// TwinCAT 3 PLC project Untitled1
// ProgramVersion: 3.1.4026.1+972e9c44872ad038b353624a861fd7e3244e9f75
// libraries:
//   Tc2_Standard, * (Beckhoff Automation GmbH)
//   Tc2_System, * (Beckhoff Automation GmbH)
//   Tc2_Utilities, * (Beckhoff Automation GmbH)
// project tree:
//   GVLs/ GVL.TcGVL
//   / PlcTask.TcTTO
//   POUs/ MAIN.TcPOU, ReadingFile.TcPOU, WritingFile.TcPOU
// real-time tasks:
//   TASK PlcTask: cycle T#10ms, priority 20, ADS port 350

CONFIGURATION Untitled1
    RESOURCE PLC ON TwinCAT3
        TASK PlcTask(INTERVAL := T#10ms, PRIORITY := 20);
        PROGRAM MAIN WITH PlcTask : MAIN;
    END_RESOURCE
END_CONFIGURATION

// ---- GVLs/GVL.TcGVL
{attribute 'qualified_only'}
VAR_GLOBAL
	sPath : STRING := 'C:\SampleFile\Test.txt';
	
END_VAR

// ---- POUs/MAIN.TcPOU
PROGRAM MAIN
VAR
	
END_VAR

ReadingFile();
WritingFile();

END_PROGRAM

// ---- POUs/ReadingFile.TcPOU
PROGRAM ReadingFile
VAR
	fbFileOpen : FB_FileOpen;
	fbFileRead : FB_FileRead;
	fbFileClose : FB_FileClose;
	hFile : UINT;
	sRead : T_MAXSTRING;
	bStartRead : BOOL;
	bReset : BOOL;
	
	eState : (init, FileOpen, FileRead, FileClose, TextFileToString , StringToINT , Error);
	i : INT;
	
	NewLineCount : INT;
	sTemp : ARRAY[1..MAX_LENGTH] OF STRING;
	nINT : ARRAY[1..MAX_LENGTH] OF INT;
	nTemp : INT;
END_VAR

VAR CONSTANT
	MAX_LENGTH : INT := 20;
END_VAR

CASE eState OF
	init :
		IF bStartRead THEN
			bStartRead := FALSE;
			eState := FileOpen;
		END_IF
		
	FileOpen :
		fbFileOpen(
			sPathName:= GVL.sPath, 
			nMode:= FOPEN_MODEREAD OR FOPEN_MODETEXT, 
			bExecute:= TRUE, 
			hFile=> hFile);
		IF NOT fbFileOpen.bBusy THEN
			IF fbFileOpen.bError THEN
				eState := Error;
			ELSE
				eState := FileRead;
				MEMSET(ADR(sRead), 0, SIZEOF(sRead) );
			END_IF
			fbFileOpen(bExecute := FALSE);
		END_IF
		
	FileRead : //fbFileRead로 값을 읽어 sRead에 값을 입력
		fbFileRead(
			hFile:= hFile, 
			pReadBuff:=ADR(sRead) , 
			cbReadLen:= SIZEOF(sRead), 
			bExecute:= TRUE);
		IF NOT fbFileRead.bBusy THEN
			IF fbFileRead.bError THEN
				eState := Error;
			ELSE
				eState := FileClose;
			END_IF
			fbFileRead(bExecute := FALSE);
		END_IF
	
	FileClose :
		fbFileClose(
			hFile:= hFile, 
			bExecute:= TRUE);
		IF NOT fbFileClose.bBusy THEN
			IF fbFileClose.bError THEN
				eState := Error;
			ELSE
				eState := TextFileToString;
			END_IF
			fbFileClose(bExecute := false);
		END_IF
	
	TextFileToString: //sRead에서 $N을 기준으로 값들을 나누고 sTemp에 각각 값을 넣음  
		MEMSET(ADR(sTemp), 0, SIZEOF(sTemp));
		FOR i:=0 TO SIZEOF(sRead) - 2 BY 1 DO
			IF sRead[i] = 10 THEN //$N
				NewLineCount := NewLineCount + 1;
				sTemp[NewLineCount] := MID(sRead,i - nTemp , nTemp + 1);
				nTemp := i+1;
			END_IF
		END_FOR
		nTemp := 0;
		NewLineCount := 0;
		eState := StringToINT;		
		
	StringToINT: //String인 sTemp값을 INT값으로 바꿔 nINT에 넣음 
		FOR i:=1 TO MAX_LENGTH BY 1 DO
			nINT[i] := STRING_TO_INT(sTemp[i]);
		END_FOR
		eState := init;
		
	Error :
		IF bReset THEN
			bReset := FALSE;
			eState := init;
		END_IF
END_CASE

END_PROGRAM

// ---- POUs/WritingFile.TcPOU
PROGRAM WritingFile
VAR
	fbFileOpen : FB_FileOpen;
	fbFileWrite : FB_FileWrite;
	fbFileClose : FB_FileClose;
	sWrite : T_MAXSTRING := '1$N22$N33$N1234$N';
	(*  $N = LF -> NewLine (줄바꾸기) *)
	hFile : UINT;
 	
	bStartWrite : BOOL;
	bReset : BOOL;
	
	eState : (init, FileOpen, FileWrite, FileClose, Error);
END_VAR

CASE eState OF
	Init:
		IF bStartWrite THEN
			bStartWrite := FALSE;
			eState := FileOpen;
		END_IF
		
	FileOpen:
		fbFileOpen(
					sNetId:= , 
					sPathName:= GVL.sPath, 
					nMode:= FOPEN_MODEWRITE OR FOPEN_MODETEXT, 
					bExecute:= TRUE,  
					hFile=> hFile);
		IF NOT fbFileOpen.bBusy THEN
			IF fbFileOpen.bError THEN
				eState := Error;
			ELSE
				eState := FileWrite;
			END_IF
			fbFileOpen(bExecute := FALSE);	
		END_IF
		
	FileWrite:
		fbFileWrite(
			hFile:= hFile, 
			pWriteBuff:= ADR(sWrite), 
			cbWriteLen:= SIZEOF(sWrite), 
			bExecute:= TRUE);
		IF NOT fbFileWrite.bBusy THEN
			IF fbFileWrite.bError THEN
				eState := Error;
			ELSE
				eState := FileClose;	
			END_IF
			fbFileWrite(bExecute := FALSE);
		END_IF
		
	FileClose:
		fbFileClose(
			hFile:= hFile, 
			bExecute:= TRUE, 
			);
		IF NOT fbFileClose.bBusy THEN
			IF fbFileClose.bError THEN
				eState := Error;
			ELSE
				eState := Init;
			END_IF
			fbFileClose(bExecute := FALSE);
		END_IF
		
	Error: 
		IF bReset THEN
			eState := init;
			bReset := FALSE;
		END_IF
END_CASE

END_PROGRAM
